// Collection that exposes only immutable methods and properties of a collection that implements I_Array.
{attribute 'enable_dynamic_creation'}
FUNCTION_BLOCK FB_Immutable_Array IMPLEMENTS I_Immutable_Array
VAR_INPUT
	ipArray : I_Array;
END_VAR
VAR
END_VAR

// Number of items in the collection.
PROPERTY _Count : T_Capacity
GET
IF THIS^.ipArray = 0 THEN RETURN; END_IF
_Count := THIS^.ipArray._Count;
END_GET
END_PROPERTY

// Checks if collection is empty.
PROPERTY _Empty : BOOL
GET
IF THIS^.ipArray = 0 THEN _Empty := TRUE; RETURN; END_IF
_Empty := THIS^.ipArray._Empty;
END_GET
END_PROPERTY

// Error status of the collection.
PROPERTY _Error_Status : T_Error
GET
IF THIS^.ipArray = 0 THEN 
	_Error_Status := GVL_Errors.ERR_INVALID_INTERFACE;
	RETURN; 
	END_IF
_Error_Status := THIS^.ipArray._Error_Status;
END_GET
END_PROPERTY

// Checks if item is contained in list.
METHOD Contains : BOOL
VAR_INPUT
	Item : ANY; // Item to find in list
END_VAR
IF THIS^.ipArray = 0 THEN RETURN; END_IF

Contains := THIS^.ipArray.Contains(Item);
END_METHOD

// Gets item from array at specified location without removing it.
METHOD Get : I_Immutable_Array
VAR_INPUT
	Index : T_Position; // Location of item
	Item : ANY;  // Variable to store returned item
END_VAR
VAR_OUTPUT
	bSuccess : BOOL;
END_VAR
Get := THIS^;

IF THIS^.ipArray = 0 THEN RETURN; END_IF

THIS^.ipArray.Get(Index, Item, bSuccess => bSuccess);
END_METHOD

// Returns item as a string, if type to string conversion is supported.
METHOD Get_As_String : I_Immutable_Array
VAR_INPUT
	Index : T_Position; // Location of item
	sItem : REFERENCE TO STRING; // Variable to store returned item.
END_VAR
VAR_OUTPUT
	bSuccess : BOOL;
END_VAR
Get_As_String := THIS^;

IF THIS^.ipArray = 0 THEN RETURN; END_IF

THIS^.ipArray.Get_As_String(Index, sItem, bSuccess => bSuccess);
END_METHOD

// Gets the type of the item at specified location.
METHOD Get_Type_At : I_Immutable_Array
VAR_INPUT
	Index : T_Position;
END_VAR
VAR_OUTPUT
	Item_Type : T_Type := T_Type.TYPE_NONE;
	bSuccess : BOOL;
END_VAR
Get_Type_At := THIS^;

IF THIS^.ipArray = 0 THEN RETURN; END_IF

THIS^.ipArray.Get_Type_At(Index, Item_Type => Item_Type, bSuccess => bSuccess);
END_METHOD

// Find the location of an item in list.
METHOD Search : I_Immutable_Array
VAR_INPUT
	Item : ANY; // Item to find in list
END_VAR
VAR_OUTPUT
	Index : T_Position := -1; //Location of item in list 
	bSuccess : BOOL;
END_VAR
Search := THIS^;

IF THIS^.ipArray = 0 THEN RETURN; END_IF

THIS^.ipArray.Search(Item, Index => Index, bSuccess => bSuccess);
END_METHOD

END_FUNCTION_BLOCK

(* stored: Version 1.1.0.1
   POU FB_Immutable_Array: Id {73f571b4-60ce-0a01-0a00-4968c563837d}, SpecialFunc None
   Property _Count: Id {30f84f30-18a4-0cc7-1a47-0d61a5ae06d0}
   Get Get: Id {876eacc8-4e1f-03ef-1324-891faad904a5}
   Property _Empty: Id {7bbbc7d9-3b84-0243-17ff-f498adef2bd4}
   Get Get: Id {09d8229f-90df-00b2-0f73-d11f28cf62d0}
   Property _Error_Status: Id {2f157328-2a26-00a9-06c6-c955fbb25e32}
   Get Get: Id {37376c54-ab20-07ff-28fc-687dd6296802}
   Method Contains: Id {14b3edc0-7ad1-0a77-365e-05bfd25ae2de}
   Method Get: Id {8878b48b-5cba-0b3e-2323-520ee798b27b}
   Method Get_As_String: Id {9f9c772d-35f0-0081-3a8f-d512bc65bb2d}
   Method Get_Type_At: Id {dbad9845-3fa2-0db4-0223-3e0ba687e21c}
   Method Search: Id {9a531ecc-dafc-07b8-03c3-7df3d3becae5} *)
